% RSLogix 500 project Flip-Flop Timers.RSS, saved by version 10.00.00.00 %
PROJECT "UNTITLED"    % processor: Bul.1763 MicroLogix 1100 Series B %

PROGRAM FILES
  LAD 2   6 rungs

DATA FILES
  O0 OUTPUT  4 elements
  I1 INPUT  6 elements
  S2 STATUS  66 elements
  B3 BINARY  1 elements
  T4 TIMER  4 elements
  C5 COUNTER  1 elements
  R6 CONTROL  1 elements
  N7 INTEGER  1 elements
  F8 FLOAT  1 elements

LADDER 2
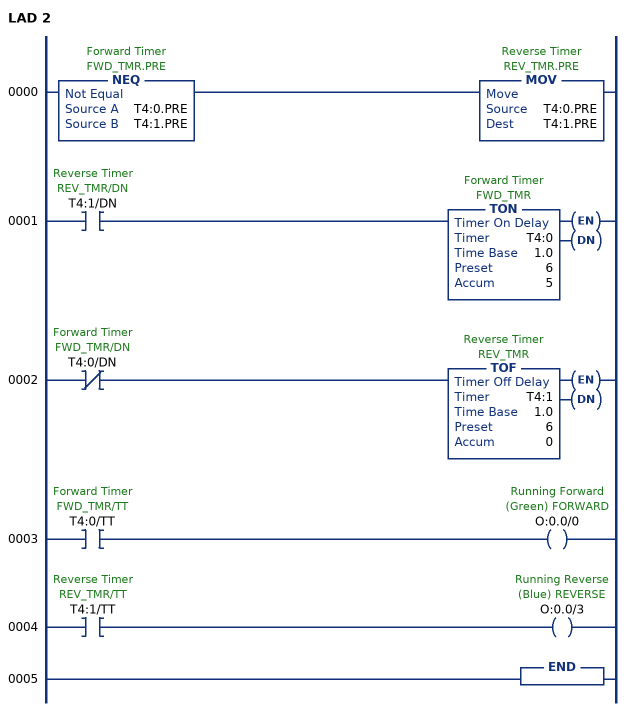
% Rung: 0 %
SOR NEQ T4:0.PRE T4:1.PRE MOV T4:0.PRE T4:1.PRE EOR
%   T4:0  FWD_TMR  "Forward Timer" %
%   T4:1  REV_TMR  "Reverse Timer" %
% Rung: 1 %
SOR XIC T4:1/DN TON T4:0 1.0 6 5 EOR
%   T4:1  REV_TMR  "Reverse Timer" %
%   T4:0  FWD_TMR  "Forward Timer" %
% Rung: 2 %
SOR XIO T4:0/DN TOF T4:1 1.0 6 0 EOR
%   T4:0  FWD_TMR  "Forward Timer" %
%   T4:1  REV_TMR  "Reverse Timer" %
% Rung: 3 %
SOR XIC T4:0/TT OTE O:0.0/0 EOR
%   T4:0  FWD_TMR  "Forward Timer" %
%   O:0.0/0  FORWARD  "Running Forward (Green)" %
% Rung: 4 %
SOR XIC T4:1/TT OTE O:0.0/3 EOR
%   T4:1  REV_TMR  "Reverse Timer" %
%   O:0.0/3  REVERSE  "Running Reverse (Blue)" %
% Rung: 5 %
SOR END EOR

OTHER DOCUMENTED ADDRESSES
  I:0.0/1  MTR_STAT  "Motor Status"

DATA TABLE (non-zero values as saved)
DATA T4
% .PRE .ACC %
% T4:0 % 6 5
% T4:1 % 6 0
% T4:3 % 3 0
